Fanuc KAREL source: kt00552.KL

PROGRAM KT00552
%STACKSIZE=65535
%PRIORITY=65535
%NOLOCKGROUP
VAR
P1 : JOINTPOS9
P2 : JOINTPOS9
OUT : JOINTPOS9
BEGIN
-- UNRESOLVED_PC line 8 opcodes [49 7E 49 7E 60 7E 4A] marker_code=0
END KT00552
